// TIA Portal project "Contadores" (V16)

(* hardware
DEVICE "S7-1200 station_1"  S7-1200 Station
   slot 0: "Rack_0"  S7-1200 Rack  Rack  V1.0
   slot 1: "PLC_1"  CPU 1214C AC/DC/Rly  6ES7 214-1BG40-0XB0  V4.4
*)

// ===== PLC "PLC_1"  CPU 1214C AC/DC/Rly =====

VAR_GLOBAL   // PLC tag table "Tabla de variables estándar"
   ""Flancos"" AT %I0.0 : Bool;
   ""Reset"" AT %I0.1 : Bool;
   ""FlancosDesc"" AT %I0.2 : Bool;
   ""ResetDesc"" AT %I0.3 : Bool;
   ""INT ASC"" AT %I0.4 : Bool;
   ""INT DESC"" AT %I0.5 : Bool;
   ""RESET TO 0"" AT %I0.6 : Bool;
   ""RESET TO 10"" AT %I0.7 : Bool;
   ""Relé"" AT %Q0.0 : Bool;
   ""OUT CTU"" AT %Q0.1 : Bool;
   ""OUT CTD"" AT %Q0.2 : Bool;
END_VAR